(* PLC project Tc2_Utilities.STRING_TO_SYSTEMTIME Demo, tc3-libraries-kb TwinCAT 3.1 *)
(* stored: creationDateTime 2026-05-10T12:00:00, modificationDateTime 2026-05-10T12:00:00 *)

PROGRAM P_Demo_STRING_TO_SYSTEMTIME
  VAR
    rResult : TIMESTRUCT;  (* STRING_TO_SYSTEMTIME 的返回值 *)
    bRun : BOOL;  (* 触发一次调用 *)
    sIn : STRING := '2024-01-01-12:00:00.000';  (* 测试用本地变量 *)
  END_VAR

            // ============================================================
// Tc2_Utilities.STRING_TO_SYSTEMTIME 演示程序（FUNCTION）
// ============================================================
// 验证步骤：
//   1. 引用 Tc2_Utilities（及类型所在依赖库 Tc2_System / Tc2_Standard）
//   2. 编译 + 登录
//   3. 强制 bRun := TRUE 一个周期
//   4. 观察 rResult 应为 TIMESTRUCT(wYear=2024, ...)
// ============================================================

IF bRun THEN
    rResult := STRING_TO_SYSTEMTIME(sIn);
    bRun := FALSE;
END_IF;

          
END_PROGRAM
